Fanuc KAREL source: COS.kl

PROGRAM T
%NOLOCKGROUP
VAR
 v0 : REAL
 res : REAL
BEGIN
 res = COS(v0)
END T
